3092:  DO[520]=(!F[574] AND F[575]) ;
3093:  DO[1871]=(F[574] AND F[575]) ;
3094:  !Einschaltdauer Einspruehen ;
3095:  TIMER[7]=((R[23])) ;
3096:  R[42]=52    ;
3097:  JMP LBL[53] ;
3098:   ;
3099:  !**************************** ;
3100:  !*        Schritt 53        * ;
3101:  !*       MS1 Reinigung      * ;
3102:  !*                          * ;
3103:  !**************************** ;
3104:   ;
3105:  LBL[53] ;
3106:  R[41]=53    ;
3107:  !MS1 Reinigung (an Pneum. Schwenk ;
3108:  F[323]=(OFF) ;
3109:  DO[2163]=(OFF) ;
3110:  DO[2164]=(OFF) ;
3111:  DO[2165]=(OFF) ;
3112:  DO[2166]=(OFF) ;
3113:  DO[2168]=(OFF) ;
3114:   ;
3115:  !Ueberwachungszeit Schwenkeinheit ;
3116:  TIMER[8]=((-7)) ;
3117:  WAIT ((TIMER[7]>=0))    ;
3118:  !MS1 Einspruehen AUS ;
3119:  DO[520]=(OFF) ;
3120:  DO[1871]=(OFF) ;
3121:  !Versetzeinheit in Ruhest. schw. ;
3122:  DO[2167]=(ON) ;
3123:  DO[2168]=(OFF) ;
3124:  !RSK Fehlerausgabe Schwenkeinheit ;
3125:  F[324]=(!DI[2164]) ;
3126:  !RSK Sammelstoerung ;
3127:  F[329]=(F[324]) ;
3128:  IF ((DI[26] OR DI[27]) AND F[324]),JMP LBL[53] ;
3129:  IF ((!F[324] OR (TIMER[8]>=0)) AND ((F[523] AND !F[524] AND DI[2161]) OR (!F[523] AND F[524] AND !DI[2162])) AND DI[2167] AND F[576]),JMP LBL[54] ;
3130:  IF ((!F[324] OR (TIMER[8]>=0)) AND ((F[523] AND !F[524] AND DI[2161]) OR (!F[523] AND F[524] AND !DI[2162])) AND !DI[2167] AND !F[576]),JMP LBL[54] ;
3131:  R[42]=53    ;
3132:   ;
3133:  !**************************** ;
3134:  !*        Schritt 54        * ;
3135:  !*       MS1 Reinigung      * ;
3136:  !* MS1 in Ruhest. schwenken * ;
3137:  !**************************** ;
3138:   ;
3139:  LBL[54] ;
3140:  R[41]=54    ;
3141:  DO[2167]=(OFF) ;
3142:  !Steuerluft EIN ;
3143:  DO[2161]=(ON) ;
3144:  !Schwenkeinheit 1 in Ruhestellung ;
3145:  DO[2163]=(!DI[2163]) ;
3146:  DO[2164]=(OFF) ;
3147:  !FRG Bewegung EIN ;
3148:  DO[2165]=(OFF) ;
3149:  DO[2166]=(!DI[2163]) ;
3150:  DO[18181]=(ON) ;
3151:  WAIT (!DI[2164] AND DI[2163])    ;
3152:  DO[18181]=(OFF) ;
3153:  !RSK Fehlerausgabe Schwenkeinheit ;
3154:  F[323]=((!DI[2163] AND (TIMER[8]>=0)) OR F[323]) ;
3155:  !RSK Sammelstoerung ;
3156:  F[329]=(F[323]) ;
3157:  DO[2163]=(OFF) ;
3158:  DO[2164]=(OFF) ;
3159:  !FRG Bewegung AUS ;
3160:  DO[2166]=(OFF) ;
3161:  IF (F[323] AND (DI[26] OR DI[27])),JMP LBL[47] ;
3162:  DO[18181]=(ON) ;
3163:  WAIT (!F[323] AND DI[2165])    ;
3164:  DO[18181]=(OFF) ;
3165:  F[323]=(OFF) ;
3166:  F[329]=(OFF) ;
3167:  !FRG in Endlage halten ein ;
3168:  DO[2165]=(ON) ;
3169:  DO[18181]=(ON) ;
3170:  WAIT   2.00(sec) ;
3171:  WAIT (!DI[2165])    ;
3172:  DO[18181]=(OFF) ;
3173:  !Steuerluft AUS ;
3174:  DO[2161]=(OFF) ;
3175:  !FRG in Endlage halten AUS ;
3176:  DO[2165]=(OFF) ;
3177:  !MS1 Zaehler ruecksetzen ;
3178:  R[21]=0    ;
3179:  !MS1 FRG Reinigung ;
3180:  F[603]=(OFF) ;
3181:  !MS1 Reinigung FK ;
3182:  F[605]=(ON) ;
3183:  R[42]=54    ;
3184:  JMP LBL[1] ;
3185:   ;
3186:  !************************** ;
3187:  !*       Schritt 55       * ;
3188:  !*      STAT EZ1/SP1      * ;
3189:  !* 2.Setzhub nach Fraesen * ;
3190:  !************************** ;
3191:   ;
3192:  LBL[55] ;
3193:  R[41]=55    ;
3194:  !RSK gestartet ;
3195:  F[321]=(OFF) ;
3196:  !EZ1/SK1 Prog. ;
3197:  IF (F[78]),GO[1]=(61) ;
3198:  IF (F[78]),GO[3]=(61) ;
3199:  WAIT    .10(sec) ;
3200:  !EZ1/SP1 schliessen ;
3201:  DO[717]=(OFF) ;
3202:  DO[718]=(ON) ;
3203:  TIMER[9]=((-8)) ;
3204:  !EZ1/SP1 Kraft erreicht ;
3205:  WAIT ((DI[718] AND !DI[717]) OR (TIMER[9]>=0))    ;
3206:  DO[18181]=((TIMER[9]>=0)) ;
3207:  WAIT (DI[718] AND !DI[717])    ;
3208:  DO[18181]=(OFF) ;
3209:  WAIT   1.00(sec) ;
3210:  !EZ1/SP1 oeffnen ;
3211:  DO[718]=(OFF) ;
3212:  DO[717]=(!DI[717]) ;
3213:  TIMER[9]=((-8)) ;
3214:  WAIT (DI[717] OR (TIMER[9]>=0))    ;
3215:  DO[18181]=((TIMER[9]>=0)) ;
3216:  WAIT (DI[717])    ;
3217:  DO[18181]=(OFF) ;
3218:  DO[717]=(OFF) ;
3219:  R[42]=55    ;
3220:  JMP LBL[16] ;
3221:   ;
3222:  !************************** ;
3223:  !*       Schritt 56       * ;
3224:  !*      STAT EZ2/SP2      * ;
3225:  !* 2.Setzhub nach Fraesen * ;
3226:  !************************** ;
3227:   ;
3228:  LBL[56] ;
3229:  R[41]=56    ;
3230:  !RSK gestartet ;
3231:  F[321]=(OFF) ;
3232:  !EZ2/SK2 Prog. ;
3233:  IF (F[285] AND F[138]),GO[3]=(65) ;
3234:  IF (!F[285] AND F[138]),GO[4]=(61) ;
3235:  IF (!F[285] AND F[138]),GO[6]=(61) ;
3236:  WAIT    .10(sec) ;
3237:  !EZ2/SP2 schliessen ;
3238:  DO[877]=(OFF) ;
3239:  DO[878]=(ON) ;
3240:  TIMER[9]=((-8)) ;
3241:  !EZ2/SP2 Kraft erreicht ;
3242:  WAIT ((DI[878] AND !DI[877]) OR (TIMER[9]>=0))    ;
3243:  DO[18181]=((TIMER[9]>=0)) ;
3244:  WAIT (DI[878] AND !DI[877])    ;
3245:  DO[18181]=(OFF) ;
3246:  WAIT   1.00(sec) ;
3247:  !EZ2/SP2 oeffnen ;
3248:  DO[878]=(OFF) ;
3249:  DO[877]=(!DI[877]) ;
3250:  TIMER[9]=((-8)) ;
3251:  WAIT (DI[877] OR (TIMER[9]>=0))    ;
3252:  DO[18181]=((TIMER[9]>=0)) ;
3253:  WAIT (DI[877])    ;
3254:  DO[18181]=(OFF) ;
3255:  DO[877]=(OFF) ;
3256:  R[42]=56    ;
3257:  JMP LBL[25] ;
3258:   ;
3259:  !************************** ;
3260:  !*       Schritt 57       * ;
3261:  !*      STAT EZ3/SP3      * ;
3262:  !* 2.Setzhub nach Fraesen * ;
3263:  !************************** ;
3264:   ;
3265:  LBL[57] ;
3266:  R[41]=57    ;
3267:  !RSK gestartet ;
3268:  F[321]=(OFF) ;
3269:  !EZ1/SK1 Prog. ;
3270:  IF (F[174]),GO[7]=(61) ;
3271:  IF (F[174]),GO[9]=(61) ;
3272:  WAIT    .10(sec) ;
3273:  !EZ3/SP3 schliessen ;
3274:  DO[1037]=(OFF) ;
3275:  DO[1038]=(ON) ;
3276:  TIMER[9]=((-8)) ;
3277:  !EZ3/SP3 Kraft erreicht ;
3278:  WAIT ((DI[1038] AND !DI[1037]) OR (TIMER[9]>=0))    ;
3279:  DO[18181]=((TIMER[9]>=0)) ;
3280:  WAIT (DI[1038] AND !DI[1037])    ;
3281:  DO[18181]=(OFF) ;
3282:  WAIT   1.00(sec) ;
3283:  !EZ3/SP3 oeffnen ;
3284:  DO[1038]=(OFF) ;
3285:  DO[1037]=(!DI[1037]) ;
3286:  TIMER[9]=((-8)) ;
3287:  WAIT (DI[1037] OR (TIMER[9]>=0))    ;
3288:  DO[18181]=((TIMER[9]>=0)) ;
3289:  WAIT (DI[1037])    ;
3290:  DO[18181]=(OFF) ;
3291:  DO[1037]=(OFF) ;
3292:  R[42]=57    ;
3293:  JMP LBL[34] ;
3294:   ;
3295:  !*************************** ;
3296:  !*************************** ;
3297:  !* Fraesen Rob EZ1 SZ1-SZ4 * ;
3298:  !*          an KF2         * ;
3299:  !*************************** ;
3300:  !*************************** ;
3301:   ;
3302:   ;
3303:  !**************************** ;
3304:  !*        Schritt 58        * ;
3305:  !* Rob EZ1 SZ1-SZ4 Auswert. * ;
3306:  !**************************** ;
3307:   ;
3308:  LBL[58] ;
3309:  R[41]=58    ;
3310:  !RSK gestartet ;
3311:  F[321]=(OFF) ;
3312:  GO[1]=(31) ;
3313:  IF (F[64]),GO[3]=(31) ;
3314:  IF (F[65]),GO[3]=(32) ;
3315:  IF (F[66]),GO[3]=(33) ;
3316:  IF (F[67]),GO[3]=(34) ;
3317:  WAIT    .10(sec) ;
3318:  DO[116]=(ON) ;
3319:  DO[130]=(ON) ;
3320:  DO[718]=(OFF) ;
3321:  DO[717]=(!DI[717]) ;
3322:  DO[18181]=(ON) ;
3323:  WAIT (DI[717])    ;
3324:  DO[18181]=(OFF) ;
3325:  DO[717]=(OFF) ;
3326:  !Anwahl Startfraesen ;
3327:  IF (F[90] AND F[78] AND !F[79]),R[41]=59 ;
3328:  !Anwahl Normalfraesen ;
3329:  IF (F[90] AND !F[78] AND F[79]),R[41]=61 ;
3330:  R[42]=58    ;
3331:  JMP LBL[R[41]] ;
3332:   ;
3333:  !***************************** ;
3334:  !*         Schritt 59        * ;
3335:  !* Rob EZ1 SZ1-SZ4 SF Teil 1 * ;
3336:  !***************************** ;
3337:   ;
3338:  LBL[59] ;
3339:  R[41]=59    ;
3340:  !RSK gestartet ;
3341:  F[321]=(OFF) ;
3342:  F[329]=(OFF) ;
3343:  F[325]=(OFF) ;
3344:  DO[718]=(OFF) ;
3345:  DO[717]=(!DI[717]) ;
3346:  DO[18181]=(ON) ;
3347:  WAIT (DI[717])    ;
3348:  DO[18181]=(OFF) ;
3349:  DO[994]=(ON) ;
3350:  DO[717]=(OFF) ;
3351:  !Warte Fraeser laeuft ;
3352:  TIMER[7]=((-3)) ;
3353:  WAIT (!DI[994] OR (TIMER[7]>=0))    ;
3354:  WAIT (DI[994] OR (TIMER[7]>=0))    ;
3355:  F[322]=((TIMER[7]>=0)) ;
3356:  DO[18181]=(ON) ;
3357:  WAIT (!DI[994])    ;
3358:  WAIT (DI[994])    ;
3359:  DO[18181]=(OFF) ;
3360:  F[322]=(OFF) ;
3361:  !EZ1/SP1 schliessen ;
3362:  DO[718]=(ON) ;
3363:  TIMER[9]=((-4)) ;
3364:  !EZ1/SP1 Kraft erreicht ;
3365:  WAIT ((DI[718] AND !DI[772] AND !DI[780] AND !DI[774] AND !DI[775]) OR (TIMER[9]>=0))    ;
3366:  DO[18181]=(ON) ;
3367:  DO[718]=((TIMER[9]<0)) ;
3368:  DO[994]=((TIMER[9]<0)) ;
3369:  WAIT ((DI[718] AND !DI[772] AND !DI[780] AND !DI[774] AND !DI[775]) OR DI[26] OR DI[27])    ;
3370:  F[325]=(DI[26] OR DI[27]) ;
3371:  DO[18181]=(OFF) ;
3372:  !EZ1/SP1 Fehler Kraftaufbau ;
3373:  IF (F[325]),JMP LBL[5906] ;
3374:  TIMER[9]=((-5)) ;
3375:  LBL[5900] ;
3376:  WAIT (!DI[994] OR F[325] OR (TIMER[9]>=0))    ;
3377:  WAIT (DI[994] OR F[325] OR (TIMER[9]>=0))    ;
3378:  R[1]=(R[1]+1) ;
3379:  F[329]=((TIMER[9]>=0)) ;
3380:  !Fraeszeit ueberschritten ;
3381:  IF (F[329]),JMP LBL[5906] ;
3382:  IF (F[64]),JMP LBL[5902] ;
3383:  IF (F[65]),JMP LBL[5903] ;
3384:  IF (F[66]),JMP LBL[5904] ;
3385:  IF (F[67]),JMP LBL[5905] ;
3386:  !Umdrehungen Vergl.SZ1 ;
3387:  LBL[5902] ;
3388:  !Umdrehungen Vergleichen ;
3389:  IF (R[1]<R[2]),JMP LBL[5900] ;
3390:  JMP LBL[5901] ;
3391:  !Umdrehungen Vergl.SZ2 ;
3392:  LBL[5903] ;
3393:  !Umdrehungen Vergleichen ;
3394:  IF (R[1]<R[8]),JMP LBL[5900] ;
3395:  JMP LBL[5901] ;
3396:  !Umdrehungen Vergl.SZ3 ;
3397:  LBL[5904] ;
3398:  !Umdrehungen Vergleichen ;
3399:  IF (R[1]<R[11]),JMP LBL[5900] ;
3400:  JMP LBL[5901] ;
3401:  !Umdrehungen Vergl.SZ4 ;
3402:  LBL[5905] ;
3403:  !Umdrehungen Vergleichen ;
3404:  IF (R[1]<R[14]),JMP LBL[5900] ;
3405:  JMP LBL[5901] ;
3406:  LBL[5901] ;
3407:  IF (F[64]),F[94]=(ON) ;
3408:  IF (F[65]),F[100]=(ON) ;
3409:  IF (F[66]),F[106]=(ON) ;
3410:  IF (F[67]),F[112]=(ON) ;
3411:  LBL[5906] ;
3412:  DO[994]=((TIMER[9]<0)) ;
3413:  !Fraeser ausblasen EIN ;
3414:  DO[995]=((TIMER[9]<0)) ;
3415:  DO[718]=(OFF) ;
3416:  !EZ1/SP1 oeffnen ;
3417:  DO[717]=(!DI[717]) ;
3418:  DO[18181]=(F[329]) ;
3419:  WAIT (!F[329] OR DI[26] OR DI[27])    ;
3420:  DO[18181]=(OFF) ;
3421:  DO[18181]=(ON) ;
3422:  WAIT (DI[717])    ;
3423:  DO[18181]=(OFF) ;
3424:  DO[717]=(OFF) ;
3425:  !Umdrehungen ruecksetzen ;
3426:  R[1]=0    ;
3427:  R[42]=59    ;
3428:  IF (F[329] OR F[325]),JMP LBL[59] ;
3429:  JMP LBL[60] ;
3430:   ;
3431:  !***************************** ;
3432:  !*         Schritt 60        * ;
3433:  !* Rob EZ1 SZ1-SZ4 SF Teil 2 * ;
3434:  !***************************** ;
3435:   ;
3436:  LBL[60] ;
3437:  R[41]=60    ;
3438:  !RSK gestartet ;
3439:  F[321]=(OFF) ;
3440:  F[329]=(OFF) ;
3441:  F[325]=(OFF) ;
3442:  DO[718]=(OFF) ;
3443:  DO[717]=(!DI[717]) ;
3444:  DO[18181]=(ON) ;
3445:  WAIT (DI[717])    ;
3446:  DO[18181]=(OFF) ;
3447:  DO[994]=(ON) ;
3448:  DO[717]=(OFF) ;
3449:  !EZ1/SP1 schliessen ;
3450:  DO[718]=(ON) ;
3451:  !Fraeser ausblasen AUS ;
3452:  DO[995]=(OFF) ;
3453:  TIMER[9]=((-4)) ;
3454:  !EZ1/SP1 Kraft erreicht ;
3455:  WAIT ((DI[718] AND !DI[772] AND !DI[780] AND !DI[774] AND !DI[775]) OR (TIMER[9]>=0))    ;
3456:  DO[18181]=(ON) ;
3457:  DO[718]=((TIMER[9]<0)) ;
3458:  DO[994]=((TIMER[9]<0)) ;
3459:  WAIT ((DI[718] AND !DI[772] AND !DI[780] AND !DI[774] AND !DI[775]) OR DI[26] OR DI[27])    ;
3460:  F[325]=(DI[26] OR DI[27]) ;
3461:  DO[18181]=(OFF) ;
3462:  !EZ1/SP1 Fehler Kraftaufbau ;
3463:  IF (F[325]),JMP LBL[60] ;
3464:  TIMER[9]=((-5)) ;
3465:  LBL[6000] ;
3466:  WAIT (!DI[994] OR F[325] OR (TIMER[9]>=0))    ;
3467:  WAIT (DI[994] OR F[325] OR (TIMER[9]>=0))    ;
3468:  R[1]=(R[1]+1) ;
3469:  F[329]=((TIMER[9]>=0)) ;
3470:  !Fraeszeit ueberschritten ;
3471:  IF (F[329]),JMP LBL[6006] ;
3472:  IF (F[64]),JMP LBL[6002] ;
3473:  IF (F[65]),JMP LBL[6003] ;
3474:  IF (F[66]),JMP LBL[6004] ;
3475:  IF (F[67]),JMP LBL[6005] ;
3476:  !Umdrehungen Vergl.SZ1 ;
3477:  LBL[6002] ;
3478:  !Umdrehungen Vergleichen ;
3479:  IF (R[1]<R[3]),JMP LBL[6000] ;
3480:  JMP LBL[6001] ;
3481:  !Umdrehungen Vergl.SZ2 ;
3482:  LBL[6003] ;
3483:  !Umdrehungen Vergleichen ;
3484:  IF (R[1]<R[9]),JMP LBL[6000] ;
3485:  JMP LBL[6001] ;
3486:  !Umdrehungen Vergl.SZ3 ;
3487:  LBL[6004] ;
3488:  !Umdrehungen Vergleichen ;
3489:  IF (R[1]<R[12]),JMP LBL[6000] ;
3490:  JMP LBL[6001] ;
3491:  !Umdrehungen Vergl.SZ4 ;
3492:  LBL[6005] ;
3493:  !Umdrehungen Vergleichen ;
3494:  IF (R[1]<R[15]),JMP LBL[6000] ;
3495:  JMP LBL[6001] ;
3496:  LBL[6001] ;
3497:  IF (F[64]),F[96]=(ON) ;
3498:  IF (F[65]),F[102]=(ON) ;
3499:  IF (F[66]),F[108]=(ON) ;
3500:  IF (F[67]),F[114]=(ON) ;
3501:  LBL[6006] ;
3502:  DO[994]=((TIMER[9]<0)) ;
3503:  !Fraeser ausblasen EIN ;
3504:  IF ((TIMER[9]<0)),DO[995]=PULSE,3.0sec ;
3505:  DO[718]=(OFF) ;
3506:  !EZ1/SP1 oeffnen ;
3507:  DO[717]=(!DI[717]) ;
3508:  DO[18181]=(F[329]) ;
3509:  WAIT (!F[329] OR DI[26] OR DI[27])    ;
3510:  DO[18181]=(OFF) ;
3511:  DO[18181]=(ON) ;
3512:  WAIT (DI[717])    ;
3513:  DO[18181]=(OFF) ;
3514:  DO[717]=(OFF) ;
3515:  !Umdrehungen ruecksetzen ;
3516:  R[1]=0    ;
3517:  R[42]=60    ;
3518:  IF (F[329] OR F[325]),JMP LBL[60] ;
3519:  JMP LBL[62] ;
3520:   ;
3521:  !********************** ;
3522:  !*     Schritt 61      * ;
3523:  !* Rob EZ1 SZ1-SZ4 NF * ;
3524:  !********************** ;
3525:   ;
3526:  LBL[61] ;
3527:  R[41]=61    ;
3528:  !RSK gestartet ;
3529:  F[321]=(OFF) ;
3530:  F[329]=(OFF) ;
3531:  F[325]=(OFF) ;
3532:  DO[718]=(OFF) ;
3533:  DO[717]=(!DI[717]) ;
3534:  DO[18181]=(ON) ;
3535:  WAIT (DI[717])    ;
3536:  DO[18181]=(OFF) ;
3537:  DO[994]=(ON) ;
3538:  DO[717]=(OFF) ;
3539:  !Warte Fraeser laeuft ;
3540:  TIMER[7]=((-3)) ;
3541:  WAIT (!DI[994] OR (TIMER[7]>=0))    ;
3542:  WAIT (DI[994] OR (TIMER[7]>=0))    ;
3543:  F[322]=((TIMER[7]>=0)) ;
3544:  DO[18181]=(ON) ;
3545:  WAIT (!DI[994])    ;
3546:  WAIT (DI[994])    ;
3547:  DO[18181]=(OFF) ;
3548:  F[322]=(OFF) ;
3549:  !EZ1/SP1 schliessen ;
3550:  DO[718]=(ON) ;
3551:  TIMER[9]=((-4)) ;
3552:  !EZ1/SP1 Kraft erreicht ;
3553:  WAIT ((DI[718] AND !DI[772] AND !DI[780] AND !DI[774] AND !DI[775]) OR (TIMER[9]>=0))    ;
3554:  DO[18181]=(ON) ;
3555:  DO[718]=((TIMER[9]<0)) ;
3556:  DO[994]=((TIMER[9]<0)) ;
3557:  WAIT ((DI[718] AND !DI[772] AND !DI[780] AND !DI[774] AND !DI[775]) OR DI[26] OR DI[27])    ;
3558:  F[325]=(DI[26] OR DI[27]) ;
3559:  DO[18181]=(OFF) ;
3560:  !EZ1/SP1 Fehler Kraftaufbau ;
3561:  IF (F[325]),JMP LBL[61] ;
3562:  TIMER[9]=((-5)) ;
3563:  LBL[6100] ;
3564:  WAIT (!DI[994] OR F[325] OR (TIMER[9]>=0))    ;
3565:  WAIT (DI[994] OR F[325] OR (TIMER[9]>=0))    ;
3566:  R[1]=(R[1]+1) ;
3567:  F[329]=((TIMER[9]>=0)) ;
3568:  !Fraeszeit ueberschritten ;
3569:  IF (F[329]),JMP LBL[6106] ;
3570:  IF (F[64]),JMP LBL[6102] ;
3571:  IF (F[65]),JMP LBL[6103] ;
3572:  IF (F[66]),JMP LBL[6104] ;
3573:  IF (F[67]),JMP LBL[6105] ;
3574:  !Umdrehungen Vergl.SZ1 ;
3575:  LBL[6102] ;
3576:  !Umdrehungen Vergleichen ;
3577:  IF (R[1]<R[4]),JMP LBL[6100] ;
3578:  JMP LBL[6101] ;
3579:  !Umdrehungen Vergl.SZ2 ;
3580:  LBL[6103] ;
3581:  !Umdrehungen Vergleichen ;
3582:  IF (R[1]<R[10]),JMP LBL[6100] ;
3583:  !Umdrehungen Vergl.SZ3 ;
3584:  LBL[6104] ;
3585:  !Umdrehungen Vergleichen ;
3586:  IF (R[1]<R[13]),JMP LBL[6100] ;
3587:  JMP LBL[6101] ;
3588:  !Umdrehungen Vergl.SZ4 ;
3589:  LBL[6105] ;
3590:  !Umdrehungen Vergleichen ;
3591:  IF (R[1]<R[16]),JMP LBL[6100] ;
3592:  LBL[6101] ;
3593:  !EZ1/SP1 2 Huebe bei NF ;
3594:  IF (!F[130]),JMP LBL[6106] ;
3595:  IF (F[98]),F[96]=(ON) ;
3596:  IF (F[104]),F[96]=(ON) ;
3597:  IF (F[110]),F[96]=(ON) ;
3598:  IF (F[116]),F[96]=(ON) ;
3599:  IF (F[64]),F[98]=(ON) ;
3600:  IF (F[65]),F[104]=(ON) ;
3601:  IF (F[66]),F[110]=(ON) ;
3602:  IF (F[67]),F[116]=(ON) ;
3603:  LBL[6106] ;
3604:  DO[994]=((TIMER[9]<0)) ;
3605:  !Fraeser ausblasen EIN ;
3606:  IF ((TIMER[9]<0)),DO[995]=PULSE,3.0sec ;
3607:  DO[718]=(OFF) ;
3608:  !EZ1/SP1 oeffnen ;
3609:  DO[717]=(!DI[717]) ;
3610:  DO[18181]=(F[329]) ;
3611:  WAIT (!F[329] OR DI[26] OR DI[27])    ;
3612:  DO[18181]=(OFF) ;
3613:  DO[18181]=(ON) ;
3614:  WAIT (DI[717])    ;
3615:  DO[18181]=(OFF) ;
3616:  DO[717]=(OFF) ;
3617:  !Umdrehungen ruecksetzen ;
3618:  R[1]=0    ;
3619:  R[42]=61    ;
3620:  IF (F[329] OR (!F[96] AND F[130])),JMP LBL[61] ;
3621:  IF (F[64]),F[98]=(ON) ;
3622:  IF (F[65]),F[104]=(ON) ;
3623:  IF (F[66]),F[110]=(ON) ;
3624:  IF (F[67]),F[116]=(ON) ;
3625:  JMP LBL[62] ;
3626:   ;
3627:  !******************************* ;
3628:  !*         Schritt 62          * ;
3629:  !* Rob EZ1 SZ1-SZ4 i.O./n.i.O. * ;
3630:  !******************************* ;
3631:   ;
3632:  LBL[62] ;
3633:  R[41]=62    ;
3634:  !Fraesueberwachung starten ;
3635:  IF (F[64]),JMP LBL[6201] ;
3636:  IF (F[65]),JMP LBL[6202] ;
3637:  IF (F[66]),JMP LBL[6203] ;
3638:  IF (F[67]),JMP LBL[6204] ;
3639:  LBL[6201] ;
3640:  TIMER[7]=((-3)) ;
3641:  WAIT (F[64] AND ((F[79] AND F[98]) OR (F[78] AND F[94] AND F[96])) OR (TIMER[7]>=0))    ;
3642:  F[329]=((TIMER[7]>=0)) ;
3643:  DO[18181]=(ON) ;
3644:  WAIT (F[64] AND ((F[79] AND F[98]) OR (F[78] AND F[94] AND F[96])))    ;
3645:  DO[18181]=(OFF) ;
3646:  JMP LBL[6200] ;
3647:  LBL[6202] ;
3648:  TIMER[7]=((-3)) ;
3649:  WAIT (F[65] AND ((F[79] AND F[104]) OR (F[78] AND F[100] AND F[102])) OR (TIMER[7]>=0))    ;
3650:  F[329]=((TIMER[7]>=0)) ;
3651:  DO[18181]=(ON) ;
3652:  WAIT (F[65] AND ((F[79] AND F[104]) OR (F[78] AND F[100] AND F[102])))    ;
3653:  DO[18181]=(OFF) ;
3654:  JMP LBL[6200] ;
3655:  LBL[6203] ;
3656:  TIMER[7]=((-3)) ;
3657:  WAIT (F[66] AND ((F[79] AND F[110]) OR (F[78] AND F[106] AND F[108])) OR (TIMER[7]>=0))    ;
3658:  F[329]=((TIMER[7]>=0)) ;
3659:  DO[18181]=(ON) ;
3660:  WAIT (F[66] AND ((F[79] AND F[110]) OR (F[78] AND F[106] AND F[108])))    ;
3661:  DO[18181]=(OFF) ;
3662:  JMP LBL[6200] ;
3663:  LBL[6204] ;
3664:  TIMER[7]=((-3)) ;
3665:  WAIT (F[67] AND ((F[79] AND F[116]) OR (F[78] AND F[112] AND F[114])) OR (TIMER[7]>=0))    ;
3666:  F[329]=((TIMER[7]>=0)) ;
3667:  DO[18181]=(ON) ;
3668:  WAIT (F[67] AND ((F[79] AND F[116]) OR (F[78] AND F[112] AND F[114])))    ;
3669:  DO[18181]=(OFF) ;
3670:  JMP LBL[6200] ;
3671:  LBL[6200] ;
3672:  R[41]=63    ;
3673:  !KF1 U-Merker ruecksetzen ;
3674:  F[94]=(OFF) ;
3675:  F[96]=(OFF) ;
3676:  F[98]=(OFF) ;
3677:  F[100]=(OFF) ;
3678:  F[102]=(OFF) ;
3679:  F[104]=(OFF) ;
3680:  F[106]=(OFF) ;
3681:  F[108]=(OFF) ;
3682:  F[110]=(OFF) ;
3683:  F[112]=(OFF) ;
3684:  F[114]=(OFF) ;
3685:  F[116]=(OFF) ;
3686:  R[42]=62    ;
3687:  JMP LBL[R[41]] ;
3688:   ;
3689:  !***************************** ;
3690:  !*        Schritt 63         * ;
3691:  !* Rob EZ1 SZ1-SZ4 Quitt SK1 * ;
3692:  !***************************** ;
3693:   ;
3694:  LBL[63] ;
3695:  R[41]=63    ;
3696:  !RSK gestartet ;
3697:  F[321]=(OFF) ;
3698:  IF (F[64]),GO[3]=1 ;
3699:  IF (F[65]),GO[3]=2 ;
3700:  IF (F[66]),GO[3]=3 ;
3701:  IF (F[67]),GO[3]=4 ;
3702:  WAIT    .10(sec) ;
3703:  DO[786]=(!F[830] AND DO[786]) ;
3704:  DO[722]=(F[830] AND DO[722]) ;
3705:  DO[116]=(OFF) ;
3706:  DO[130]=(OFF) ;
3707:  DO[18181]=(ON) ;
3708:  WAIT ((!DI[786] AND DI[787] AND !DI[788]) OR F[830])    ;
3709:  WAIT ((!DI[722] AND DI[724] AND !DI[723] OR F[329]) OR !F[830])    ;
3710:  !FK Fraesen ;
3711:  F[91]=((!DI[786] AND DI[787] AND !DI[788] AND !F[830]) OR (!DI[722] AND DI[724] AND !DI[723] AND F[830]) AND !F[322] AND !F[325] AND !F[329]) ;
3712:  DO[18181]=(OFF) ;
3713:  DO[786]=(!F[830] AND DO[786]) ;
3714:  DO[722]=(F[830] AND DO[722]) ;
3715:  R[42]=63    ;
3716:  JMP LBL[1] ;
3717:   ;
3718:  !*************************** ;
3719:  !*************************** ;
3720:  !* Fraesen Rob EZ1 SZ1-SZ4 * ;
3721:  !*          an KF3         * ;
3722:  !*************************** ;
3723:  !*************************** ;
3724:   ;
3725:   ;
3726:  !**************************** ;
3727:  !*        Schritt 64        * ;
3728:  !* Rob EZ1 SZ1-SZ4 Auswert. * ;
3729:  !**************************** ;
3730:   ;
3731:  LBL[64] ;
3732:  R[41]=64    ;
3733:  !RSK gestartet ;
3734:  F[321]=(OFF) ;
3735:  GO[1]=(31) ;
3736:  IF (F[64]),GO[3]=(31) ;
3737:  IF (F[65]),GO[3]=(32) ;
3738:  IF (F[66]),GO[3]=(33) ;
3739:  IF (F[67]),GO[3]=(34) ;
3740:  WAIT    .10(sec) ;
3741:  DO[116]=(ON) ;
3742:  DO[130]=(ON) ;
3743:  DO[718]=(OFF) ;
3744:  DO[717]=(!DI[717]) ;
3745:  DO[18181]=(ON) ;
3746:  WAIT (DI[717])    ;
3747:  DO[18181]=(OFF) ;
3748:  DO[717]=(OFF) ;
3749:  !Anwahl Startfraesen ;
3750:  IF (F[90] AND F[78] AND !F[79]),R[41]=65 ;
3751:  !Anwahl Normalfraesen ;
3752:  IF (F[90] AND !F[78] AND F[79]),R[41]=67 ;
3753:  R[42]=64    ;
3754:  JMP LBL[R[41]] ;
3755:   ;
3756:  !***************************** ;
3757:  !*         Schritt 65        * ;
3758:  !* Rob EZ1 SZ1-SZ4 SF Teil 1 * ;
3759:  !***************************** ;
3760:   ;
3761:  LBL[65] ;
3762:  R[41]=65    ;
3763:  !RSK gestartet ;
3764:  F[321]=(OFF) ;
3765:  F[329]=(OFF) ;
3766:  F[325]=(OFF) ;
3767:  DO[718]=(OFF) ;
3768:  DO[717]=(!DI[717]) ;
3769:  DO[18181]=(ON) ;
3770:  WAIT (DI[717])    ;
3771:  DO[18181]=(OFF) ;
3772:  DO[1154]=(ON) ;
3773:  DO[717]=(OFF) ;
3774:  !Warte Fraeser laeuft ;
3775:  TIMER[7]=((-3)) ;
3776:  WAIT (!DI[1154] OR (TIMER[7]>=0))    ;
3777:  WAIT (DI[1154] OR (TIMER[7]>=0))    ;
3778:  F[322]=((TIMER[7]>=0)) ;
3779:  DO[18181]=(ON) ;
3780:  WAIT (!DI[1154])    ;
3781:  WAIT (DI[1154])    ;
3782:  DO[18181]=(OFF) ;
3783:  F[322]=(OFF) ;
3784:  !EZ1/SP1 schliessen ;
3785:  DO[718]=(ON) ;
3786:  TIMER[9]=((-4)) ;
3787:  !EZ1/SP1 Kraft erreicht ;
3788:  WAIT ((DI[718] AND !DI[772] AND !DI[780] AND !DI[774] AND !DI[775]) OR (TIMER[9]>=0))    ;
3789:  DO[18181]=(ON) ;
3790:  DO[718]=((TIMER[9]<0)) ;
3791:  DO[1154]=((TIMER[9]<0)) ;
3792:  WAIT ((DI[718] AND !DI[772] AND !DI[780] AND !DI[774] AND !DI[775]) OR DI[26] OR DI[27])    ;
3793:  F[325]=(DI[26] OR DI[27]) ;
3794:  DO[18181]=(OFF) ;
3795:  !EZ1/SP1 Fehler Kraftaufbau ;
3796:  IF (F[325]),JMP LBL[6506] ;
3797:  TIMER[9]=((-5)) ;
3798:  LBL[6500] ;
3799:  WAIT (!DI[1154] OR F[325] OR (TIMER[9]>=0))    ;
3800:  WAIT (DI[1154] OR F[325] OR (TIMER[9]>=0))    ;
3801:  R[1]=(R[1]+1) ;
3802:  F[329]=((TIMER[9]>=0)) ;
3803:  !Fraeszeit ueberschritten ;
3804:  IF (F[329]),JMP LBL[6506] ;
3805:  IF (F[64]),JMP LBL[6502] ;
3806:  IF (F[65]),JMP LBL[6503] ;
3807:  IF (F[66]),JMP LBL[6504] ;
3808:  IF (F[67]),JMP LBL[6505] ;
3809:  !Umdrehungen Vergl.SZ1 ;
3810:  LBL[6502] ;
3811:  !Umdrehungen Vergleichen ;
3812:  IF (R[1]<R[2]),JMP LBL[6500] ;
3813:  JMP LBL[6501] ;
3814:  !Umdrehungen Vergl.SZ2 ;
3815:  LBL[6503] ;
3816:  !Umdrehungen Vergleichen ;
3817:  IF (R[1]<R[8]),JMP LBL[6500] ;
3818:  JMP LBL[6501] ;
3819:  !Umdrehungen Vergl.SZ3 ;
3820:  LBL[6504] ;
3821:  !Umdrehungen Vergleichen ;
3822:  IF (R[1]<R[11]),JMP LBL[6500] ;
3823:  JMP LBL[6501] ;
3824:  !Umdrehungen Vergl.SZ4 ;
3825:  LBL[6505] ;
3826:  !Umdrehungen Vergleichen ;
3827:  IF (R[1]<R[14]),JMP LBL[6500] ;
3828:  JMP LBL[6501] ;
3829:  LBL[6501] ;
3830:  IF (F[64]),F[94]=(ON) ;
3831:  IF (F[65]),F[100]=(ON) ;
3832:  IF (F[66]),F[106]=(ON) ;
3833:  IF (F[67]),F[112]=(ON) ;
3834:  LBL[6506] ;
3835:  DO[1154]=((TIMER[9]<0)) ;
3836:  !Fraeser ausblasen EIN ;
3837:  DO[1155]=((TIMER[9]<0)) ;
3838:  DO[718]=(OFF) ;
3839:  !EZ1/SP1 oeffnen ;
3840:  DO[717]=(!DI[717]) ;
3841:  DO[18181]=(F[329]) ;
3842:  WAIT (!F[329] OR DI[26] OR DI[27])    ;
3843:  DO[18181]=(OFF) ;
3844:  DO[18181]=(ON) ;
3845:  WAIT (DI[717])    ;
3846:  DO[18181]=(OFF) ;
3847:  DO[717]=(OFF) ;
3848:  !Umdrehungen ruecksetzen ;
3849:  R[1]=0    ;
3850:  R[42]=65    ;
3851:  IF (F[329] OR F[325]),JMP LBL[65] ;
3852:  JMP LBL[66] ;
3853:   ;
3854:  !***************************** ;
3855:  !*         Schritt 66        * ;
3856:  !* Rob EZ1 SZ1-SZ4 SF Teil 2 * ;
3857:  !***************************** ;
3858:   ;
3859:  LBL[66] ;
3860:  R[41]=66    ;
3861:  !RSK gestartet ;
3862:  F[321]=(OFF) ;
3863:  F[329]=(OFF) ;
3864:  F[325]=(OFF) ;
3865:  DO[718]=(OFF) ;
3866:  DO[717]=(!DI[717]) ;
3867:  DO[18181]=(ON) ;
3868:  WAIT (DI[717])    ;
3869:  DO[18181]=(OFF) ;
3870:  DO[1154]=(ON) ;
3871:  DO[717]=(OFF) ;
3872:  !EZ1/SP1 schliessen ;
3873:  DO[718]=(ON) ;
3874:  !Fraeser ausblasen AUS ;
3875:  DO[1155]=(OFF) ;
3876:  TIMER[9]=((-4)) ;
3877:  !EZ1/SP1 Kraft erreicht ;
3878:  WAIT ((DI[718] AND !DI[772] AND !DI[780] AND !DI[774] AND !DI[775]) OR (TIMER[9]>=0))    ;
3879:  DO[18181]=(ON) ;
3880:  DO[718]=((TIMER[9]<0)) ;
3881:  DO[1154]=((TIMER[9]<0)) ;
3882:  WAIT ((DI[718] AND !DI[772] AND !DI[780] AND !DI[774] AND !DI[775]) OR DI[26] OR DI[27])    ;
3883:  F[325]=(DI[26] OR DI[27]) ;
3884:  DO[18181]=(OFF) ;
3885:  !EZ1/SP1 Fehler Kraftaufbau ;
3886:  IF (F[325]),JMP LBL[66] ;
3887:  TIMER[9]=((-5)) ;
3888:  LBL[6600] ;
3889:  WAIT (!DI[1154] OR F[325] OR (TIMER[9]>=0))    ;
3890:  WAIT (DI[1154] OR F[325] OR (TIMER[9]>=0))    ;
3891:  R[1]=(R[1]+1) ;
3892:  F[329]=((TIMER[9]>=0)) ;
3893:  !Fraeszeit ueberschritten ;
3894:  IF (F[329]),JMP LBL[6606] ;
3895:  IF (F[64]),JMP LBL[6602] ;
3896:  IF (F[65]),JMP LBL[6603] ;
3897:  IF (F[66]),JMP LBL[6604] ;
3898:  IF (F[67]),JMP LBL[6605] ;
3899:  !Umdrehungen Vergl.SZ1 ;
3900:  LBL[6602] ;
3901:  !Umdrehungen Vergleichen ;
3902:  IF (R[1]<R[3]),JMP LBL[6600] ;
3903:  JMP LBL[6601] ;
3904:  !Umdrehungen Vergl.SZ2 ;
3905:  LBL[6603] ;
3906:  !Umdrehungen Vergleichen ;
3907:  IF (R[1]<R[9]),JMP LBL[6600] ;
3908:  JMP LBL[6601] ;
3909:  !Umdrehungen Vergl.SZ3 ;
3910:  LBL[6604] ;
3911:  !Umdrehungen Vergleichen ;
3912:  IF (R[1]<R[12]),JMP LBL[6600] ;
3913:  JMP LBL[6601] ;
3914:  !Umdrehungen Vergl.SZ4 ;
3915:  LBL[6605] ;
3916:  !Umdrehungen Vergleichen ;
3917:  IF (R[1]<R[15]),JMP LBL[6600] ;
3918:  JMP LBL[6601] ;
3919:  LBL[6601] ;
3920:  IF (F[64]),F[96]=(ON) ;
3921:  IF (F[65]),F[102]=(ON) ;
3922:  IF (F[66]),F[108]=(ON) ;
3923:  IF (F[67]),F[114]=(ON) ;
3924:  LBL[6606] ;
3925:  DO[1154]=((TIMER[9]<0)) ;
3926:  !Fraeser ausblasen EIN ;
3927:  IF ((TIMER[9]<0)),DO[1155]=PULSE,3.0sec ;
3928:  DO[718]=(OFF) ;
3929:  !EZ1/SP1 oeffnen ;
3930:  DO[717]=(!DI[717]) ;
3931:  DO[18181]=(F[329]) ;
3932:  WAIT (!F[329] OR DI[26] OR DI[27])    ;
3933:  DO[18181]=(OFF) ;
3934:  DO[18181]=(ON) ;
3935:  WAIT (DI[717])    ;
3936:  DO[18181]=(OFF) ;
3937:  DO[717]=(OFF) ;
3938:  !Umdrehungen ruecksetzen ;
3939:  R[1]=0    ;
3940:  R[42]=66    ;
3941:  IF (F[329] OR F[325]),JMP LBL[66] ;
3942:  JMP LBL[68] ;
3943:   ;
3944:  !********************** ;
3945:  !*     Schritt 67     * ;
3946:  !* Rob EZ1 SZ1-SZ4 NF * ;
3947:  !********************** ;
3948:   ;
3949:  LBL[67] ;
3950:  R[41]=67    ;
3951:  !RSK gestartet ;
3952:  F[321]=(OFF) ;
3953:  F[329]=(OFF) ;
3954:  F[325]=(OFF) ;
3955:  DO[718]=(OFF) ;
3956:  DO[717]=(!DI[717]) ;
3957:  DO[18181]=(ON) ;
3958:  WAIT (DI[717])    ;
3959:  DO[18181]=(OFF) ;
3960:  DO[1154]=(ON) ;
3961:  DO[717]=(OFF) ;
3962:  !Warte Fraeser laeuft ;
3963:  TIMER[7]=((-3)) ;
3964:  WAIT (!DI[1154] OR (TIMER[7]>=0))    ;
3965:  WAIT (DI[1154] OR (TIMER[7]>=0))    ;
3966:  F[322]=((TIMER[7]>=0)) ;
3967:  DO[18181]=(ON) ;
3968:  WAIT (!DI[1154])    ;
3969:  WAIT (DI[1154])    ;
3970:  DO[18181]=(OFF) ;
3971:  F[322]=(OFF) ;
3972:  !EZ1/SP1 schliessen ;
3973:  DO[718]=(ON) ;
3974:  TIMER[9]=((-4)) ;
3975:  !EZ1/SP1 Kraft erreicht ;
3976:  WAIT ((DI[718] AND !DI[772] AND !DI[780] AND !DI[774] AND !DI[775]) OR (TIMER[9]>=0))    ;
3977:  DO[18181]=(ON) ;
3978:  DO[718]=((TIMER[9]<0)) ;
3979:  DO[1154]=((TIMER[9]<0)) ;
3980:  WAIT ((DI[718] AND !DI[772] AND !DI[780] AND !DI[774] AND !DI[775]) OR DI[26] OR DI[27])    ;
3981:  F[325]=(DI[26] OR DI[27]) ;
3982:  DO[18181]=(OFF) ;
3983:  !EZ1/SP1 Fehler Kraftaufbau ;
3984:  IF (F[325]),JMP LBL[67] ;
3985:  TIMER[9]=((-5)) ;
3986:  LBL[6700] ;
3987:  WAIT (!DI[1154] OR F[325] OR (TIMER[9]>=0))    ;
3988:  WAIT (DI[1154] OR F[325] OR (TIMER[9]>=0))    ;
3989:  R[1]=(R[1]+1) ;
3990:  F[329]=((TIMER[9]>=0)) ;
3991:  !Fraeszeit ueberschritten ;
3992:  IF (F[329]),JMP LBL[6706] ;
3993:  IF (F[64]),JMP LBL[6702] ;
3994:  IF (F[65]),JMP LBL[6703] ;
3995:  IF (F[66]),JMP LBL[6704] ;
3996:  IF (F[67]),JMP LBL[6705] ;
3997:  !Umdrehungen Vergl.SZ1 ;
3998:  LBL[6702] ;
3999:  !Umdrehungen Vergleichen ;
4000:  IF (R[1]<R[4]),JMP LBL[6700] ;
4001:  JMP LBL[6701] ;
4002:  !Umdrehungen Vergl.SZ2 ;
4003:  LBL[6703] ;
4004:  !Umdrehungen Vergleichen ;
4005:  IF (R[1]<R[10]),JMP LBL[6700] ;
4006:  !Umdrehungen Vergl.SZ3 ;
4007:  LBL[6704] ;
4008:  !Umdrehungen Vergleichen ;
4009:  IF (R[1]<R[13]),JMP LBL[6700] ;
4010:  JMP LBL[6701] ;
4011:  !Umdrehungen Vergl.SZ4 ;
4012:  LBL[6705] ;
4013:  !Umdrehungen Vergleichen ;
4014:  IF (R[1]<R[16]),JMP LBL[6700] ;
4015:  LBL[6701] ;
4016:  !EZ1/SP1 2 Huebe bei NF ;
4017:  IF (!F[130]),JMP LBL[6706] ;
4018:  IF (F[98]),F[96]=(ON) ;
4019:  IF (F[104]),F[96]=(ON) ;
4020:  IF (F[110]),F[96]=(ON) ;
4021:  IF (F[116]),F[96]=(ON) ;
4022:  IF (F[64]),F[98]=(ON) ;
4023:  IF (F[65]),F[104]=(ON) ;
4024:  IF (F[66]),F[110]=(ON) ;
4025:  IF (F[67]),F[116]=(ON) ;
4026:  LBL[6706] ;
4027:  DO[1154]=((TIMER[9]<0)) ;
4028:  !Fraeser ausblasen EIN ;
4029:  IF ((TIMER[9]<0)),DO[1155]=PULSE,3.0sec ;
4030:  DO[718]=(OFF) ;
4031:  !EZ1/SP1 oeffnen ;
4032:  DO[717]=(!DI[717]) ;
4033:  DO[18181]=(F[329]) ;
4034:  WAIT (!F[329] OR DI[26] OR DI[27])    ;
4035:  DO[18181]=(OFF) ;
4036:  DO[18181]=(ON) ;
4037:  WAIT (DI[717])    ;
4038:  DO[18181]=(OFF) ;
4039:  DO[717]=(OFF) ;
4040:  !Umdrehungen ruecksetzen ;
4041:  R[1]=0    ;
4042:  R[42]=67    ;
4043:  IF (F[329] OR (!F[96] AND F[130])),JMP LBL[67] ;
4044:  IF (F[64]),F[98]=(ON) ;
4045:  IF (F[65]),F[104]=(ON) ;
4046:  IF (F[66]),F[110]=(ON) ;
4047:  IF (F[67]),F[116]=(ON) ;
4048:  JMP LBL[68] ;
4049:   ;
4050:  !******************************* ;
4051:  !*         Schritt 68           * ;
4052:  !* Rob EZ1 SZ1-SZ4 i.O./n.i.O. * ;
4053:  !******************************* ;
4054:   ;
4055:  LBL[68] ;
4056:  R[41]=68    ;
4057:  !Fraesueberwachung starten ;
4058:  IF (F[64]),JMP LBL[6801] ;
4059:  IF (F[65]),JMP LBL[6802] ;
4060:  IF (F[66]),JMP LBL[6803] ;
4061:  IF (F[67]),JMP LBL[6804] ;
4062:  LBL[6801] ;
4063:  TIMER[7]=((-3)) ;
4064:  WAIT (F[64] AND ((F[79] AND F[98]) OR (F[78] AND F[94] AND F[96])) OR (TIMER[7]>=0))    ;
4065:  F[329]=((TIMER[7]>=0)) ;
4066:  DO[18181]=(ON) ;
4067:  WAIT (F[64] AND ((F[79] AND F[98]) OR (F[78] AND F[94] AND F[96])))    ;
4068:  DO[18181]=(OFF) ;
4069:  JMP LBL[6800] ;
4070:  LBL[6802] ;
4071:  TIMER[7]=((-3)) ;
4072:  WAIT (F[65] AND ((F[79] AND F[104]) OR (F[78] AND F[100] AND F[102])) OR (TIMER[7]>=0))    ;
4073:  F[329]=((TIMER[7]>=0)) ;
4074:  DO[18181]=(ON) ;
4075:  WAIT (F[65] AND ((F[79] AND F[104]) OR (F[78] AND F[100] AND F[102])))    ;
4076:  DO[18181]=(OFF) ;
4077:  JMP LBL[6800] ;
4078:  LBL[6803] ;
4079:  TIMER[7]=((-3)) ;
4080:  WAIT (F[66] AND ((F[79] AND F[110]) OR (F[78] AND F[106] AND F[108])) OR (TIMER[7]>=0))    ;
4081:  F[329]=((TIMER[7]>=0)) ;
4082:  DO[18181]=(ON) ;
4083:  WAIT (F[66] AND ((F[79] AND F[110]) OR (F[78] AND F[106] AND F[108])))    ;
4084:  DO[18181]=(OFF) ;
4085:  JMP LBL[6800] ;
4086:  LBL[6804] ;
4087:  TIMER[7]=((-3)) ;
4088:  WAIT (F[67] AND ((F[79] AND F[116]) OR (F[78] AND F[112] AND F[114])) OR (TIMER[7]>=0))    ;
4089:  F[329]=((TIMER[7]>=0)) ;
4090:  DO[18181]=(ON) ;
4091:  WAIT (F[67] AND ((F[79] AND F[116]) OR (F[78] AND F[112] AND F[114])))    ;
4092:  DO[18181]=(OFF) ;
4093:  JMP LBL[6800] ;
4094:  LBL[6800] ;
4095:  R[41]=69    ;
4096:  !KF1 U-Merker ruecksetzen ;
4097:  F[94]=(OFF) ;
4098:  F[96]=(OFF) ;
4099:  F[98]=(OFF) ;
4100:  F[100]=(OFF) ;
4101:  F[102]=(OFF) ;
4102:  F[104]=(OFF) ;
4103:  F[106]=(OFF) ;
4104:  F[108]=(OFF) ;
4105:  F[110]=(OFF) ;
4106:  F[112]=(OFF) ;
4107:  F[114]=(OFF) ;
4108:  F[116]=(OFF) ;
4109:  R[42]=68    ;
4110:  JMP LBL[R[41]] ;
4111:   ;
4112:  !***************************** ;
4113:  !*        Schritt 69         * ;
4114:  !* Rob EZ1 SZ1-SZ4 Quitt SK1 * ;
4115:  !***************************** ;
4116:   ;
4117:  LBL[69] ;
4118:  R[41]=69    ;
4119:  !RSK gestartet ;
4120:  F[321]=(OFF) ;
4121:  IF (F[64]),GO[3]=1 ;
4122:  IF (F[65]),GO[3]=2 ;
4123:  IF (F[66]),GO[3]=3 ;
4124:  IF (F[67]),GO[3]=4 ;
4125:  WAIT    .10(sec) ;
4126:  DO[786]=(F[830] AND DO[786]) ;
4127:  DO[722]=(!F[830] AND DO[722]) ;
4128:  DO[116]=(OFF) ;
4129:  DO[130]=(OFF) ;
4130:  DO[18181]=(ON) ;
4131:  WAIT ((!DI[786] AND DI[787] AND !DI[788]) OR F[830])    ;
4132:  WAIT ((!DI[722] AND DI[724] AND !DI[723] OR F[329]) OR !F[830])    ;
4133:  !FK Fraesen ;
4134:  F[91]=((!DI[786] AND DI[787] AND !DI[788] AND !F[830]) OR (!DI[722] AND DI[724] AND !DI[723] AND F[830]) AND !F[322] AND !F[325] AND !F[329]) ;
4135:  DO[18181]=(OFF) ;
4136:  DO[786]=(!F[830]) ;
4137:  DO[722]=(F[830]) ;
4138:  R[42]=69    ;
4139:  JMP LBL[1] ;
4140:   ;
4141:  !********************** ;
4142:  !*     Schritt 70     * ;
4143:  !* ROB STP1 SZ1 Start * ;
4144:  !********************** ;
4145:   ;
4146:  LBL[70] ;
4147:  R[41]=70    ;
4148:  !RSK gestartet ;
4149:  F[321]=(OFF) ;
4150:  F[122]=(OFF) ;
4151:  F[322]=(OFF) ;
4152:  F[323]=(OFF) ;
4153:  F[324]=(OFF) ;
4154:  F[325]=(OFF) ;
4155:  F[329]=(OFF) ;
4156:  !Rob. STP1 SZ1 beim Fraesen ;
4157:  DO[116]=(ON) ;
4158:  DO[130]=(ON) ;
4159:  !Anwahl Startfraesen ;
4160:  IF (F[90] AND F[78] AND !F[79]),R[41]=71 ;
4161:  !Anwahl Normalfraesen ;
4162:  IF (F[90] AND !F[78] AND F[79]),R[41]=73 ;
4163:  R[42]=70    ;
4164:  JMP LBL[R[41]] ;
4165:   ;
4166:  !************************** ;
4167:  !*      Schritt 71        * ;
4168:  !* Rob STP1 SZ1 SF Teil 1 * ;
4169:  !************************** ;
4170:   ;
4171:  LBL[71] ;
4172:  R[41]=71    ;
4173:  !RSK gestartet ;
4174:  F[321]=(OFF) ;
4175:  F[329]=(OFF) ;
4176:  F[325]=(OFF) ;
4177:  !KF1 einschalten ;
4178:  DO[864]=(ON) ;
4179:  !Warte Fraeser laeuft ;
4180:  TIMER[7]=((-3)) ;
4181:  WAIT (!DI[864] OR (TIMER[7]>=0))    ;
4182:  WAIT (DI[864] OR (TIMER[7]>=0))    ;
4183:  F[322]=((TIMER[7]>=0)) ;
4184:  DO[18181]=(ON) ;
4185:  WAIT (!DI[864])    ;
4186:  WAIT (DI[864])    ;
4187:  DO[18181]=(OFF) ;
4188:  F[322]=(OFF) ;
4189:  !KF1 hochfahren ;
4190:  DO[863]=(ON) ;
4191:  TIMER[8]=((-5)) ;
4192:  WAIT (!DI[863] OR (TIMER[8]>=0))    ;
4193:  F[324]=((TIMER[8]>=0)) ;
4194:  DO[18181]=(ON) ;
4195:  WAIT (!DI[863])    ;
4196:  DO[18181]=(OFF) ;
4197:  F[324]=(OFF) ;
4198:  TIMER[9]=((-5)) ;
4199:  LBL[7100] ;
4200:  WAIT (!DI[864] OR (TIMER[9]>=0))    ;
4201:  WAIT (DI[864] OR (TIMER[9]>=0))    ;
4202:  R[1]=(R[1]+1) ;
4203:  F[329]=((TIMER[9]>=0)) ;
4204:  !Fraeszeit ueberschritten ;
4205:  IF (F[329]),JMP LBL[7103] ;
4206:  IF (F[64]),JMP LBL[7102] ;
4207:  !Umdrehungen Vergl.SZ1 ;
4208:  LBL[7102] ;
4209:  !Umdrehungen Vergleichen ;
4210:  IF (R[1]<R[2]),JMP LBL[7100] ;
4211:  JMP LBL[7101] ;
4212:  LBL[7101] ;
4213:  IF (F[64]),F[94]=(ON) ;
4214:  LBL[7103] ;
4215:  DO[864]=(OFF) ;
4216:  DO[18181]=(F[329]) ;
4217:  WAIT (!F[329] OR DI[26] OR DI[27])    ;
4218:  DO[18181]=(OFF) ;
4219:  !KF1 runterfahren ;
4220:  DO[863]=(OFF) ;
4221:  TIMER[8]=((-5)) ;
4222:  WAIT (DI[863] OR (TIMER[8]>=0))    ;
4223:  F[324]=((TIMER[8]>=0)) ;
4224:  DO[18181]=(ON) ;
4225:  WAIT (DI[863])    ;
4226:  DO[18181]=(OFF) ;
4227:  F[324]=(OFF) ;
4228:  !Umdrehungen ruecksetzen ;
4229:  R[1]=0    ;
4230:  R[42]=71    ;
4231:  IF (F[329] OR F[325]),JMP LBL[71] ;
4232:  JMP LBL[72] ;
4233:   ;
4234:  !************************** ;
4235:  !*      Schritt 72        * ;
4236:  !* Rob STP1 SZ1 SF Teil 2 * ;
4237:  !************************** ;
4238:   ;
4239:  LBL[72] ;
4240:  R[41]=72    ;
4241:  !RSK gestartet ;
4242:  F[321]=(OFF) ;
4243:  F[329]=(OFF) ;
4244:  F[325]=(OFF) ;
4245:  !KF1 einschalten ;
4246:  DO[864]=(ON) ;
4247:  !Warte Fraeser laeuft ;
4248:  TIMER[7]=((-3)) ;
4249:  WAIT (!DI[864] OR (TIMER[7]>=0))    ;
4250:  WAIT (DI[864] OR (TIMER[7]>=0))    ;
4251:  F[322]=((TIMER[7]>=0)) ;
4252:  DO[18181]=(ON) ;
4253:  WAIT (!DI[864])    ;
4254:  WAIT (DI[864])    ;
4255:  DO[18181]=(OFF) ;
4256:  F[322]=(OFF) ;
4257:  !KF1 hochfahren ;
4258:  DO[863]=(ON) ;
4259:  TIMER[8]=((-5)) ;
4260:  WAIT (!DI[863] OR (TIMER[8]>=0))    ;
4261:  F[324]=((TIMER[8]>=0)) ;
4262:  DO[18181]=(ON) ;
4263:  WAIT (!DI[863])    ;
4264:  DO[18181]=(OFF) ;
4265:  F[324]=(OFF) ;
4266:  TIMER[9]=((-5)) ;
4267:  LBL[7200] ;
4268:  WAIT (!DI[864] OR (TIMER[9]>=0))    ;
4269:  WAIT (DI[864] OR (TIMER[9]>=0))    ;
4270:  R[1]=(R[1]+1) ;
4271:  F[329]=((TIMER[9]>=0)) ;
4272:  !Fraeszeit ueberschritten ;
4273:  IF (F[329]),JMP LBL[7203] ;
4274:  IF (F[64]),JMP LBL[7202] ;
4275:  !Umdrehungen Vergl.SZ1 ;
4276:  LBL[7202] ;
4277:  !Umdrehungen Vergleichen ;
4278:  IF (R[1]<R[3]),JMP LBL[7200] ;
4279:  JMP LBL[7201] ;
4280:  LBL[7201] ;
4281:  IF (F[64]),F[96]=(ON) ;
4282:  LBL[7203] ;
4283:  DO[864]=(OFF) ;
4284:  DO[18181]=(F[329]) ;
4285:  WAIT (!F[329] OR DI[26] OR DI[27])    ;
4286:  DO[18181]=(OFF) ;
4287:  !KF1 runterfahren ;
4288:  DO[863]=(OFF) ;
4289:  TIMER[8]=((-5)) ;
4290:  WAIT (DI[863] OR (TIMER[8]>=0))    ;
4291:  F[324]=((TIMER[8]>=0)) ;
4292:  DO[18181]=(ON) ;
4293:  WAIT (DI[863])    ;
4294:  DO[18181]=(OFF) ;
4295:  F[324]=(OFF) ;
4296:  !Umdrehungen ruecksetzen ;
4297:  R[1]=0    ;
4298:  R[42]=73    ;
4299:  IF (F[329] OR F[325]),JMP LBL[72] ;
4300:  JMP LBL[73] ;
4301:   ;
4302:   ;
4303:  !******************* ;
4304:  !*   Schritt 73    * ;
4305:  !* Rob STP1 SZ1 NF * ;
4306:  !******************* ;
4307:   ;
4308:  LBL[73] ;
4309:  R[41]=73    ;
4310:  !RSK gestartet ;
4311:  F[321]=(OFF) ;
4312:  F[329]=(OFF) ;
4313:  F[325]=(OFF) ;
4314:  !KF1 einschalten ;
4315:  DO[864]=(ON) ;
4316:  !Warte Fraeser laeuft ;
4317:  TIMER[7]=((-3)) ;
4318:  WAIT (!DI[864] OR (TIMER[7]>=0))    ;
4319:  WAIT (DI[864] OR (TIMER[7]>=0))    ;
4320:  F[322]=((TIMER[7]>=0)) ;
4321:  DO[18181]=(ON) ;
4322:  WAIT (!DI[864])    ;
4323:  WAIT (DI[864])    ;
4324:  DO[18181]=(OFF) ;
4325:  F[322]=(OFF) ;
4326:  !KF1 hochfahren ;
4327:  DO[863]=(ON) ;
4328:  TIMER[8]=((-5)) ;
4329:  WAIT (!DI[863] OR (TIMER[8]>=0))    ;
4330:  F[324]=((TIMER[8]>=0)) ;
4331:  DO[18181]=(ON) ;
4332:  WAIT (!DI[863])    ;
4333:  DO[18181]=(OFF) ;
4334:  F[324]=(OFF) ;
4335:  TIMER[9]=((-5)) ;
4336:  LBL[7300] ;
4337:  WAIT (!DI[864] OR (TIMER[9]>=0))    ;
4338:  WAIT (DI[864] OR (TIMER[9]>=0))    ;
4339:  R[1]=(R[1]+1) ;
4340:  F[329]=((TIMER[9]>=0)) ;
4341:  !Fraeszeit ueberschritten ;
4342:  IF (F[329]),JMP LBL[7303] ;
4343:  IF (F[64]),JMP LBL[7302] ;
4344:  !Umdrehungen Vergl.SZ1 ;
4345:  LBL[7302] ;
4346:  !Umdrehungen Vergleichen ;
4347:  IF (R[1]<R[4]),JMP LBL[7300] ;
4348:  JMP LBL[7301] ;
4349:  LBL[7301] ;
4350:  IF (F[64]),F[98]=(ON) ;
4351:  LBL[7303] ;
4352:  DO[864]=(OFF) ;
4353:  DO[18181]=(F[329]) ;
4354:  WAIT (!F[329] OR DI[26] OR DI[27])    ;
4355:  DO[18181]=(OFF) ;
4356:  !KF1 runterfahren ;
4357:  DO[863]=(OFF) ;
4358:  TIMER[8]=((-5)) ;
4359:  WAIT (DI[863] OR (TIMER[8]>=0))    ;
4360:  F[324]=((TIMER[8]>=0)) ;
4361:  DO[18181]=(ON) ;
4362:  WAIT (DI[863])    ;
4363:  DO[18181]=(OFF) ;
4364:  F[324]=(OFF) ;
4365:  !Umdrehungen ruecksetzen ;
4366:  R[1]=0    ;
4367:  R[42]=72    ;
4368:  IF (F[329] OR F[325]),JMP LBL[73] ;
4369:  JMP LBL[74] ;
4370:   ;
4371:  !*************************** ;
4372:  !*       Schritt 74        * ;
4373:  !* Rob STP SZ1 i.O./n.i.O. * ;
4374:  !*************************** ;
4375:   ;
4376:  LBL[74] ;
4377:  R[41]=74    ;
4378:  !Fraesueberwachung starten ;
4379:  TIMER[7]=((-3)) ;
4380:  WAIT (F[64] AND ((F[79] AND F[98]) OR (F[78] AND F[94] AND F[96])) OR (TIMER[7]>=0))    ;
4381:  F[329]=((TIMER[7]>=0)) ;
4382:  DO[18181]=(ON) ;
4383:  WAIT (F[64] AND ((F[79] AND F[98]) OR (F[78] AND F[94] AND F[96])))    ;
4384:  DO[18181]=(OFF) ;
4385:  R[41]=75    ;
4386:  !KF1 U-Merker ruecksetzen ;
4387:  F[94]=(OFF) ;
4388:  F[96]=(OFF) ;
4389:  F[98]=(OFF) ;
4390:  R[42]=74    ;
4391:  JMP LBL[R[41]] ;
4392:   ;
4393:  !***************************** ;
4394:  !*        Schritt 75         * ;
4395:  !*   Rob STP SZ1 Quitt SK1   * ;
4396:  !***************************** ;
4397:   ;
4398:  LBL[75] ;
4399:  R[41]=75    ;
4400:  !RSK gestartet ;
4401:  F[321]=(OFF) ;
4402:  IF (F[64] AND !F[329]),GO[3]=1 ;
4403:  WAIT    .10(sec) ;
4404:  DO[786]=(!F[329] AND !F[322]) ;
4405:  DO[18181]=(ON) ;
4406:  WAIT ((!DI[786] AND DI[787] AND !DI[788] AND !F[329]) OR DI[26] OR DI[27])    ;
4407:  !FK Fraesen ;
4408:  F[91]=(!F[329]) ;
4409:  DO[18181]=(OFF) ;
4410:  DO[786]=(OFF) ;
4411:  DO[116]=(OFF) ;
4412:  DO[130]=(OFF) ;
4413:  R[41]=1    ;
4414:  IF (!F[329]),JMP LBL[7500] ;
4415:  R[41]=70    ;
4416:  LBL[7500] ;
4417:  R[42]=75    ;
4418:  JMP LBL[R[41]] ;
4419:   ;
4420:  !***************************** ;
4421:  !*        Schritt 76         * ;
4422:  !*       ROB STP1 SZ1        * ;
4423:  !*   Start mit Braeuer KF/KW * ;
4424:  !***************************** ;
4425:   ;
4426:  LBL[76] ;
4427:  R[41]=76    ;
4428:  !RSK gestartet ;
4429:  F[122]=(OFF) ;
4430:  F[321]=(OFF) ;
4431:  F[322]=(OFF) ;
4432:  F[323]=(OFF) ;
4433:  F[324]=(OFF) ;
4434:  F[325]=(OFF) ;
4435:  F[329]=(OFF) ;
4436:  GO[1]=(31) ;
4437:  IF (F[64]),GO[3]=(31) ;
4438:  WAIT    .10(sec) ;
4439:  !Hilfsflags Funktionstest KF Moto ;
4440:  !F[312]=(OFF) ;
4441:  !F[313]=(OFF) ;
4442:  !Rob. STP1 SZ1 beim Fraesen ;
4443:  DO[116]=(ON) ;
4444:  DO[130]=(ON) ;
4445:  !Rob. STP1 öffnen ;
4446:  DO[718]=(OFF) ;
4447:  DO[717]=(!DI[717]) ;
4448:  DO[18181]=(ON) ;
4449:  WAIT (DI[717])    ;
4450:  DO[18181]=(OFF) ;
4451:  DO[717]=(OFF) ;
4452:  !Anwahl Startfraesen ;
4453:  IF (F[90] AND F[78] AND !F[79]),R[41]=77 ;
4454:  !Anwahl Normalfraesen ;
4455:  IF (F[90] AND !F[78] AND F[79]),R[41]=79 ;
4456:  R[42]=76    ;
4457:  JMP LBL[R[41]] ;
4458:   ;
4459:  !************************** ;
4460:  !*      Schritt 77        * ;
4461:  !* Rob STP1 SZ1 SF Teil 1 * ;
4462:  !************************** ;
4463:   ;
4464:  LBL[77] ;
4465:  R[41]=77    ;
4466:  !RSK gestartet ;
4467:  F[321]=(OFF) ;
4468:  F[329]=(OFF) ;
4469:  F[325]=(OFF) ;
4470:  !Rob. STP1 öffnen ;
4471:  DO[718]=(OFF) ;
4472:  DO[717]=(!DI[717]) ;
4473:  DO[18181]=(ON) ;
4474:  WAIT (DI[717])    ;
4475:  DO[18181]=(OFF) ;
4476:  DO[717]=(OFF) ;
4477:  !KF1 / Ausblasen einschalten ;
4478:  R[1]=0    ;
4479:  DO[834]=(!F[289]) ;
4480:  DO[835]=(!F[289]) ;
4481:  DO[858]=(F[289]) ;
4482:  DO[859]=(F[289]) ;
4483:  !Warte Fraeser laeuft ;
4484:  TIMER[7]=((-3)) ;
4485:  !Funktionstest Fraeser laeuft ;
4486:  !F[312]=(ON) ;
4487:  !F[313]=(R[1]>2) ;
4488:  WAIT ((!DI[858] AND DI[863] AND F[289]) OR (!DI[834] AND !F[289]) OR (TIMER[7]>=0))    ;
4489:  WAIT ((DI[858] AND DI[863] AND !F[289]) OR (DI[834] AND !F[289]) OR (TIMER[7]>=0))    ;
4490:  F[322]=((TIMER[7]>=0)) ;
4491:  DO[18181]=(ON) ;
4492:  WAIT (DI[858] AND DI[863])    ;
4493:  DO[18181]=(OFF) ;
4494:  F[322]=(OFF) ;
4495:  !Rob. STP1 schliessen ;
4496:  DO[717]=(OFF) ;
4497:  DO[720]=(DI[717]) ;
4498:  DO[718]=(ON) ;
4499:  TIMER[11]=((-3)) ;
4500:  DO[720]=(TIMER[11]>=0) ;
4501:  TIMER[9]=((-4)) ;
4502:  !STP1 Kraft erreicht ;
4503:  WAIT ((DI[718] AND !DI[772] AND !DI[780] AND !DI[774] AND !DI[775]) OR (TIMER[9]>=0))    ;
4504:  DO[18181]=(ON) ;
4505:  DO[718]=((TIMER[9]<0)) ;
4506:  DO[834]=((TIMER[9]<0)) ;
4507:  DO[858]=((TIMER[9]<0)) ;
4508:  WAIT ((DI[718] AND !DI[772] AND !DI[780] AND !DI[774] AND !DI[775]) OR DI[26] OR DI[27])    ;
4509:  F[325]=(DI[26] OR DI[27]) ;
4510:  DO[18181]=(OFF) ;
4511:  !STP1 Fehler Kraftaufbau ;
4512:  IF (F[325]),JMP LBL[406] ;
4513:  TIMER[9]=((-5)) ;
4514:  LBL[7710] ;
4515:  WAIT ((!DI[858] AND DI[863] AND F[289]) OR (!DI[834] AND !F[289]) OR (TIMER[9]>=0))    ;
4516:  WAIT ((DI[858] AND DI[863] AND F[289]) OR (DI[834] AND !F[289]) OR (TIMER[9]>=0))    ;
4517:  R[1]=(R[1]+1) ;
4518:  F[329]=((TIMER[9]>=0)) ;
4519:  !Fraeszeit ueberschritten ;
4520:  IF (F[329]),JMP LBL[7713] ;
4521:  IF (F[64]),JMP LBL[7712] ;
4522:  !Umdrehungen Vergl. STP1 ;
4523:  LBL[7712] ;
4524:  !Umdrehungen Vergleichen ;
4525:  IF (R[1]<R[2]),JMP LBL[7710] ;
4526:  JMP LBL[7711] ;
4527:  LBL[7711] ;
4528:  IF (F[64]),F[94]=(ON) ;
4529:  LBL[7713] ;
4530:  DO[834]=((TIMER[9]<0)) ;
4531:  DO[858]=((TIMER[9]<0)) ;
4532:  !Fraeser ausblasen EIN ;
4533:  DO[835]=((TIMER[9]<0)) ;
4534:  DO[859]=((TIMER[9]<0)) ;
4535:  DO[718]=(OFF) ;
4536:  !EZ1/SP1 oeffnen ;
4537:  DO[718]=(OFF) ;
4538:  DO[717]=(!DI[717]) ;
4539:  DO[18181]=(F[329]) ;
4540:  WAIT (!F[329] OR DI[26] OR DI[27])    ;
4541:  DO[18181]=(OFF) ;
4542:  DO[18181]=(ON) ;
4543:  WAIT (DI[717])    ;
4544:  DO[18181]=(OFF) ;
4545:  DO[717]=(OFF) ;
4546:  !Umdrehungen ruecksetzen ;
4547:  R[1]=0    ;
4548:  R[42]=77    ;
4549:  IF (F[329] OR F[325]),JMP LBL[77] ;
4550:  JMP LBL[78] ;
4551:   ;
4552:  !************************** ;
4553:  !*      Schritt 78        * ;
4554:  !* Rob STP1 SZ1 SF Teil 2 * ;
4555:  !************************** ;
4556:   ;
4557:  LBL[78] ;
4558:  R[41]=78    ;
4559:  !RSK gestartet ;
4560:  F[321]=(OFF) ;
4561:  F[329]=(OFF) ;
4562:  F[325]=(OFF) ;
4563:  !Rob. STP1 öffnen ;
4564:  DO[718]=(OFF) ;
4565:  DO[717]=(!DI[717]) ;
4566:  DO[18181]=(ON) ;
4567:  WAIT (DI[717])    ;
4568:  DO[18181]=(OFF) ;
4569:  DO[717]=(OFF) ;
4570:  !Rob. STP1 schliessen ;
4571:  DO[717]=(OFF) ;
4572:  DO[720]=(DI[717]) ;
4573:  DO[718]=(ON) ;
4574:  TIMER[11]=((-3)) ;
4575:  DO[720]=(TIMER[11]>=0) ;
4576:  !KF1 / Ausblasen einschalten ;
4577:  DO[834]=(!F[329]) ;
4578:  DO[835]=(!F[329]) ;
4579:  DO[858]=(F[329]) ;
4580:  DO[859]=(F[329]) ;
4581:  TIMER[9]=((-4)) ;
4582:  !STP1 Kraft erreicht ;
4583:  WAIT ((DI[718] AND !DI[772] AND !DI[780] AND !DI[774] AND !DI[775]) OR (TIMER[9]>=0))    ;
4584:  DO[18181]=(ON) ;
4585:  DO[718]=((TIMER[9]<0)) ;
4586:  DO[834]=((TIMER[9]<0)) ;
4587:  DO[858]=((TIMER[9]<0)) ;
4588:  WAIT ((DI[718] AND !DI[772] AND !DI[780] AND !DI[774] AND !DI[775]) OR DI[26] OR DI[27])    ;
4589:  F[325]=(DI[26] OR DI[27]) ;
4590:  DO[18181]=(OFF) ;
4591:  !STP1 Fehler Kraftaufbau ;
4592:  IF (F[325]),JMP LBL[78] ;
4593:  TIMER[9]=((-5)) ;
4594:  LBL[7810] ;
4595:  WAIT ((!DI[858] AND DI[863] AND F[289]) OR (!DI[834] AND !F[289]) OR (TIMER[9]>=0))    ;
4596:  WAIT ((DI[858] AND DI[863] AND F[289]) OR (DI[834] AND !F[289]) OR (TIMER[9]>=0))    ;
4597:  R[1]=(R[1]+1) ;
4598:  F[329]=((TIMER[9]>=0)) ;
4599:  !Fraeszeit ueberschritten ;
4600:  IF (F[329]),JMP LBL[7813] ;
4601:  IF (F[64]),JMP LBL[7812] ;
4602:  !Umdrehungen Vergl. STP1 ;
4603:  LBL[7812] ;
4604:  !Umdrehungen Vergleichen ;
4605:  IF (R[1]<R[2]),JMP LBL[7810] ;
4606:  JMP LBL[7811] ;
4607:  LBL[7811] ;
4608:  IF (F[64]),F[94]=(ON) ;
4609:  LBL[7813] ;
4610:  DO[834]=((TIMER[9]<0)) ;
4611:  DO[858]=((TIMER[9]<0)) ;
4612:  !Fraeser ausblasen EIN ;
4613:  DO[835]=PULSE,4.0sec ;
4614:  DO[859]=PULSE,4.0sec ;
4615:  DO[718]=(OFF) ;
4616:  !EZ1/SP1 oeffnen ;
4617:  DO[718]=(OFF) ;
4618:  DO[717]=(!DI[717]) ;
4619:  DO[18181]=(F[329]) ;
4620:  WAIT (!F[329] OR DI[26] OR DI[27])    ;
4621:  DO[18181]=(OFF) ;
4622:  DO[18181]=(ON) ;
4623:  WAIT (DI[717])    ;
4624:  DO[18181]=(OFF) ;
4625:  DO[717]=(OFF) ;
4626:  !Umdrehungen ruecksetzen ;
4627:  R[1]=0    ;
4628:  R[42]=78    ;
4629:  IF (F[329] OR F[325]),JMP LBL[78] ;
4630:  JMP LBL[79] ;
4631:   ;
4632:  !******************* ;
4633:  !*   Schritt 79   * ;
4634:  !* Rob STP1 SZ1 NF * ;
4635:  !******************* ;
4636:   ;
4637:  LBL[79] ;
4638:  R[41]=79    ;
4639:  !RSK gestartet ;
4640:  F[321]=(OFF) ;
4641:  F[329]=(OFF) ;
4642:  F[325]=(OFF) ;
4643:  !Zähler wegspeichern für 2ten Hub ;
4644:  R[45]=(R[4]) ;
4645:  IF (F[98] AND F[732]),R[4]=(R[43]) ;
4646:  !Rob. STP1 öffnen ;
4647:  DO[718]=(OFF) ;
4648:  DO[717]=(!DI[717]) ;
4649:  DO[18181]=(ON) ;
4650:  WAIT (DI[717])    ;
4651:  DO[18181]=(OFF) ;
4652:  DO[717]=(OFF) ;
4653:  !KF1 / Ausblasen einschalten ;
4654:  R[1]=0    ;
4655:  DO[834]=(!F[329]) ;
4656:  DO[835]=(!F[329]) ;
4657:  DO[858]=(!F[329]) ;
4658:  DO[859]=(!F[329]) ;
4659:  !Warte Fraeser laeuft ;
4660:  TIMER[7]=((-3)) ;
4661:  WAIT ((!DI[858] AND DI[863] AND F[289]) OR (!DI[834] AND !F[289]) OR (TIMER[7]>=0))    ;
4662:  WAIT ((DI[858] AND DI[863] AND F[289]) OR (DI[834] AND !F[289]) OR (TIMER[7]>=0))    ;
4663:  F[322]=((TIMER[7]>=0)) ;
4664:  DO[18181]=(ON) ;
4665:  WAIT ((!DI[858] AND DI[863] AND F[289]) OR (!DI[834] AND !F[289]))    ;
4666:  WAIT ((DI[858] AND DI[863] AND F[289]) OR (DI[834] AND !F[289]))    ;
4667:  DO[18181]=(OFF) ;
4668:  F[322]=(OFF) ;
4669:  !Rob. STP1 schliessen ;
4670:  DO[717]=(OFF) ;
4671:  DO[720]=(DI[717]) ;
4672:  DO[718]=(ON) ;
4673:  TIMER[11]=((-3)) ;
4674:  DO[720]=(TIMER[11]>=0) ;
4675:  TIMER[9]=((-4)) ;
4676:  !STP1 Kraft erreicht ;
4677:  WAIT ((DI[718] AND !DI[772] AND !DI[780] AND !DI[774] AND !DI[775]) OR (TIMER[9]>=0))    ;
4678:  DO[18181]=(ON) ;
4679:  DO[718]=((TIMER[9]<0)) ;
4680:  DO[834]=((TIMER[9]<0)) ;
4681:  DO[858]=((TIMER[9]<0)) ;
4682:  WAIT ((DI[718] AND !DI[772] AND !DI[780] AND !DI[774] AND !DI[775]) OR DI[26] OR DI[27])    ;
4683:  F[325]=(DI[26] OR DI[27]) ;
4684:  DO[18181]=(OFF) ;
4685:  !STP1 Fehler Kraftaufbau ;
4686:  IF (F[325]),JMP LBL[79] ;
4687:  TIMER[9]=((-5)) ;
4688:  LBL[7910] ;
4689:  WAIT ((!DI[858] AND DI[863] AND F[289]) OR (!DI[834] AND !F[289]) OR (TIMER[9]>=0))    ;
4690:  WAIT ((DI[858] AND DI[863] AND F[289]) OR (DI[834] AND !F[289]) OR (TIMER[9]>=0))    ;
4691:  R[1]=(R[1]+1) ;
4692:  F[329]=((TIMER[9]>=0)) ;
4693:  !Fraeszeit ueberschritten ;
4694:  IF (F[329]),JMP LBL[7913] ;
4695:  IF (F[64]),JMP LBL[7912] ;
4696:  !Umdrehungen Vergl. STP1 ;
4697:  LBL[7912] ;
4698:  !Umdrehungen Vergleichen ;
4699:  IF (R[1]<R[4]),JMP LBL[7910] ;
4700:  !Umdrehungen Vergleichen ;
4701:  IF (R[1]<R[13]),JMP LBL[7910] ;
4702:  JMP LBL[7911] ;
4703:  LBL[7911] ;
4704:  !EZ1/SP1 2 Huebe bei NF ;
4705:  IF (!F[130]),JMP LBL[7913] ;
4706:  IF (F[98]),F[96]=(ON) ;
4707:  IF (F[104]),F[96]=(ON) ;
4708:  IF (F[110]),F[96]=(ON) ;
4709:  IF (F[116]),F[96]=(ON) ;
4710:  IF (F[64]),F[98]=(ON) ;
4711:  IF (F[65]),F[104]=(ON) ;
4712:  IF (F[66]),F[110]=(ON) ;
4713:  IF (F[67]),F[116]=(ON) ;
4714:  LBL[7913] ;
4715:  DO[834]=((TIMER[9]<0)) ;
4716:  DO[858]=((TIMER[9]<0)) ;
4717:  !Fraeser ausblasen EIN ;
4718:  !Fraeser ausblasen EIN ;
4719:  DO[835]=PULSE,4.0sec ;
4720:  DO[859]=PULSE,4.0sec ;
4721:  DO[718]=(OFF) ;
4722:  !EZ1/SP1 oeffnen ;
4723:  DO[718]=(OFF) ;
4724:  DO[717]=(!DI[717]) ;
4725:  DO[18181]=(F[329]) ;
4726:  WAIT (!F[329] OR DI[26] OR DI[27])    ;
4727:  DO[18181]=(OFF) ;
4728:  DO[18181]=(ON) ;
4729:  WAIT (DI[717])    ;
4730:  DO[18181]=(OFF) ;
4731:  DO[717]=(OFF) ;
4732:  !Umdrehungen ruecksetzen ;
4733:  R[1]=0    ;
4734:  R[42]=79    ;
4735:  !Zähler umschreiben für 2ten Hub ;
4736:  IF (F[98] AND F[732] AND F[64]),GO[3]=36 ;
4737:  IF (F[104] AND F[732] AND F[65]),GO[3]=37 ;
4738:  IF (F[110] AND F[732] AND F[66]),GO[3]=38 ;
4739:  IF (F[116] AND F[732] AND F[67]),GO[3]=39 ;
4740:  IF (F[96] AND F[732]),R[4]=(R[45]) ;
4741:  !Aufruf 2ter Hub ;
4742:  IF (F[329] OR (!F[96] AND F[130])),JMP LBL[79] ;
4743:  IF (F[64]),F[98]=(ON) ;
4744:  IF (F[65]),F[104]=(ON) ;
4745:  JMP LBL[80] ;
4746:   ;
4747:  !*************************** ;
4748:  !*       Schritt 80        * ;
4749:  !* Rob STP SZ1 i.O./n.i.O. * ;
4750:  !*************************** ;
4751:   ;
4752:  LBL[80] ;
4753:  R[41]=80    ;
4754:  !Fraesueberwachung starten ;
4755:  IF (F[64]),JMP LBL[8010] ;
4756:  IF (F[65]),JMP LBL[8011] ;
4757:  IF (F[66]),JMP LBL[8012] ;
4758:  IF (F[67]),JMP LBL[8013] ;
4759:  LBL[8010] ;
4760:  TIMER[7]=((-3)) ;
4761:  WAIT (F[64] AND ((F[79] AND F[98]) OR (F[78] AND F[94] AND F[96])) OR (TIMER[7]>=0))    ;
4762:  F[329]=((TIMER[7]>=0)) ;
4763:  DO[18181]=(ON) ;
4764:  WAIT (F[64] AND ((F[79] AND F[98]) OR (F[78] AND F[94] AND F[96])))    ;
4765:  DO[18181]=(OFF) ;
4766:  JMP LBL[8013] ;
4767:  !Platzhalter für Erweiterung STPs ;
4768:  LBL[8011] ;
4769:  JMP LBL[8013] ;
4770:  !Platzhalter für Erweiterung STPs ;
4771:  LBL[8012] ;
4772:  JMP LBL[8013] ;
4773:  !Platzhalter für Erweiterung STPs ;
4774:  LBL[8013] ;
4775:  R[41]=81    ;
4776:  !KF1 U-Merker ruecksetzen ;
4777:  F[94]=(OFF) ;
4778:  F[96]=(OFF) ;
4779:  F[98]=(OFF) ;
4780:  F[100]=(OFF) ;
4781:  F[102]=(OFF) ;
4782:  F[104]=(OFF) ;
4783:  F[106]=(OFF) ;
4784:  F[108]=(OFF) ;
4785:  F[110]=(OFF) ;
4786:  F[112]=(OFF) ;
4787:  F[114]=(OFF) ;
4788:  F[116]=(OFF) ;
4789:  R[42]=80    ;
4790:  JMP LBL[R[41]] ;
4791:   ;
4792:  !***************************** ;
4793:  !*        Schritt 81         * ;
4794:  !*   Rob STP1 Quitt SK1      * ;
4795:  !***************************** ;
4796:   ;
4797:  LBL[81] ;
4798:  R[41]=81    ;
4799:  DO[717]=OFF ;
4800:  DO[858]=OFF ;
4801:  DO[859]=OFF ;
4802:  !RSK gestartet ;
4803:  F[321]=(OFF) ;
4804:  IF (F[64]),GO[3]=1 ;
4805:  IF (F[65]),GO[3]=2 ;
4806:  IF (F[66]),GO[3]=3 ;
4807:  IF (F[67]),GO[3]=4 ;
4808:  WAIT    .10(sec) ;
4809:  DO[786]=(!F[329] AND !F[322]) ;
4810:  DO[18181]=(ON) ;
4811:  WAIT ((!DI[786] AND DI[787] AND !DI[788] AND !F[329]) OR DI[26] OR DI[27])    ;
4812:  !FK Fraesen ;
4813:  F[91]=(!DI[786] AND DI[787] AND !DI[788] AND !F[322] AND !F[325] AND !F[329]) ;
4814:  DO[116]=(OFF) ;
4815:  DO[130]=(OFF) ;
4816:  !FK Fraesen ;
4817:  F[91]=((!DI[786] AND DI[787] AND !DI[788] AND !F[830]) OR (!DI[722] AND DI[724] AND !DI[723] AND F[830]) AND !F[322] AND !F[325] AND !F[329]) ;
4818:  DO[18181]=(OFF) ;
4819:  R[41]=1    ;
4820:  IF (!F[329]),JMP LBL[8110] ;
4821:  R[41]=76    ;
4822:  LBL[8110] ;
4823:  R[42]=81    ;
4824:  JMP LBL[R[41]] ;
4825:  !********************** ;
4826:  !********************** ;
4827:  !* Ende Makro_Schritt * ;
4828:  !********************** ;
4829:  !********************** ;
4830:   ;
/POS
/END
